FUNCTION_BLOCK DrillModel
  (* Standard: 61499-2 *)
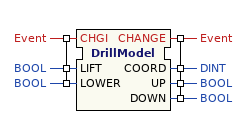
  EVENT_INPUT
    CHGI WITH LIFT, LOWER;
  END_EVENT
  EVENT_OUTPUT
    CHANGE WITH UP, DOWN, COORD;
  END_EVENT
  VAR_INPUT
    LIFT : BOOL;
    LOWER : BOOL;
  END_VAR
  VAR_OUTPUT
    COORD : DINT;
    UP : BOOL;
    DOWN : BOOL;
  END_VAR
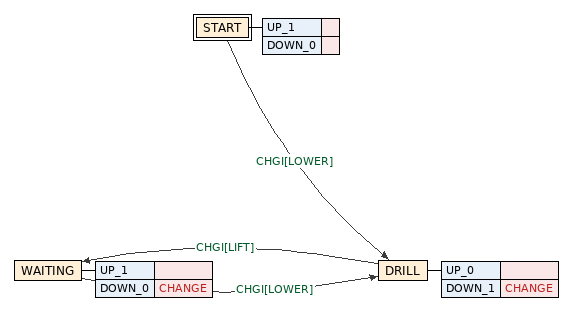
  EC_STATES
    START : UP_1, DOWN_0;
    DRILL : UP_0, DOWN_1 -> CHANGE;
    WAITING : UP_1, DOWN_0 -> CHANGE;
  END_STATES
  EC_TRANSITIONS
    START TO DRILL := CHGI[LOWER];
    DRILL TO WAITING := CHGI[LIFT];
    WAITING TO DRILL := CHGI[LOWER];
  END_TRANSITIONS
  ALGORITHM UP_0 IN ST:
UP := FALSE;&#10;
  END_ALGORITHM
  ALGORITHM UP_1 IN ST:
UP := TRUE;&#10;
  END_ALGORITHM
  ALGORITHM DOWN_0 IN ST:
DOWN := FALSE;&#10;
  END_ALGORITHM
  ALGORITHM DOWN_1 IN ST:
DOWN := TRUE;&#10;
  END_ALGORITHM
END_FUNCTION_BLOCK
